// TIA Portal V17 export
// export: Created 2022-02-03T14:45:12.3278315Z, ExportSetting WithDefaults, DisplayName Totally Integrated Automation Portal, DisplayVersion V17, DisplayName TIA Portal Openness, DisplayVersion V17, DisplayName TIA Portal Version Control Interface, DisplayVersion V17, DisplayName SINAMICS Startdrive Advanced, DisplayVersion V17, DisplayName SINAMICS Startdrive G130, G150, S120, S150, SINAMICS MV, S210, DisplayVersion V17, DisplayName SINAMICS Startdrive G110M, G120, G120C, G120D, G120P, G115D, DisplayVersion V17, DisplayName STEP 7 Professional, DisplayVersion V17, DisplayName STEP 7 Safety, DisplayVersion V17, DisplayName WinCC Advanced, DisplayVersion V17
FUNCTION_BLOCK "ConveyorWeights"   // FB4, LAD
VERSION : 0.1
// stored: Access Published, AutoNumber true, IsIECCheckEnabled false, IsRetainMemResEnabled false, MemoryReserve 100, SetENOAutomatically false, UDAEnableTagReadback false
   VAR_INPUT
      weightSimulation : UInt;
      bLightBarrier : Bool;
      conveyorLeft : Bool;
      occupiedBay : Array["FIRSTBAY".."LASTBAY"] of Bool;
   END_VAR
   VAR_OUTPUT
      weightLightBarrier : UInt;
      weightBay : Array["FIRSTBAY".."LASTBAY"] of UInt;
   END_VAR
   VAR_IN_OUT
      weightConveyor : UInt;
   END_VAR
   VAR
      statOldbLightBarrier : Bool;
      statOldOccupiedBay : Array["FIRSTBAY".."LASTBAY"] of Bool;
      InstIEC_Timer1 { S7_SetPoint := 'True'} : TON_TIME;
      InstIEC_Timer2 { S7_SetPoint := 'True'} : TON_TIME;
      InstIEC_Timer3 { S7_SetPoint := 'True'} : TON_TIME;
   END_VAR
   VAR_TEMP   // added for the SCL form of the ladder/FBD networks
      _w1 : Bool;
   END_VAR
BEGIN

REGION Network 1
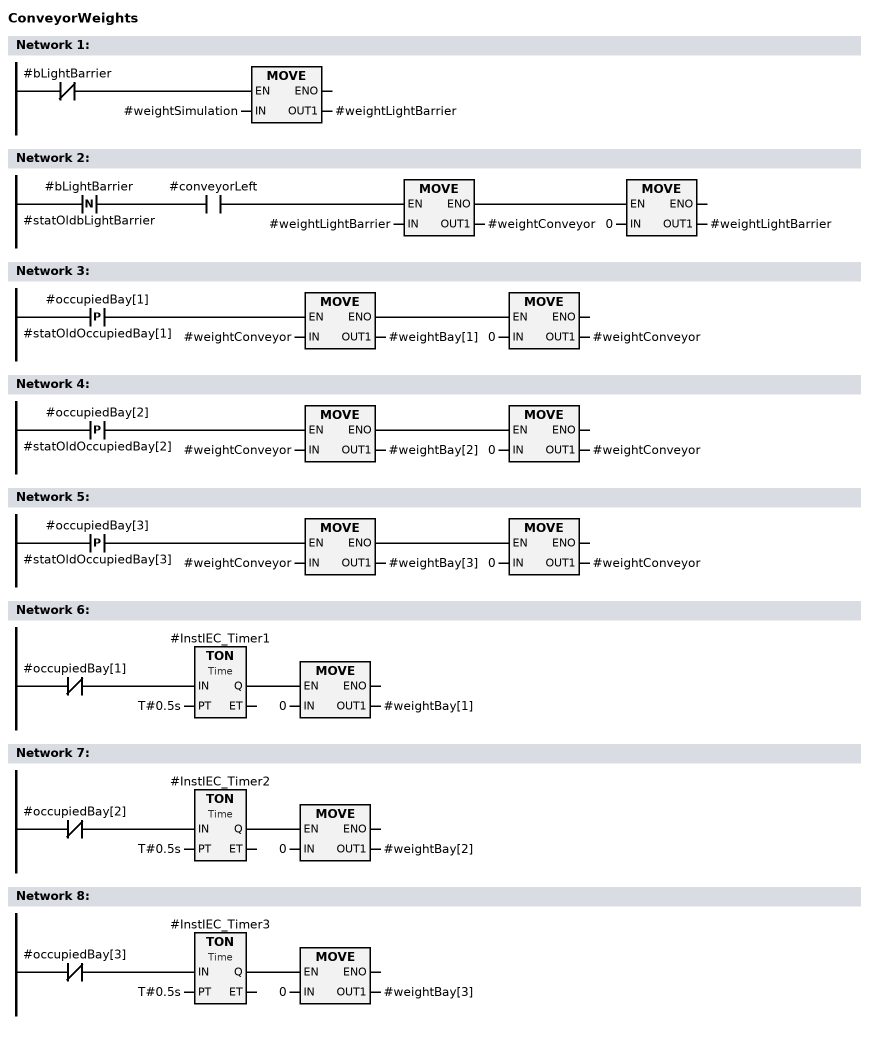
   RUNG wire#powerrail
      I_Contact( #bLightBarrier )
      Move(in := #weightSimulation, out1 => #weightLightBarrier)
   END_RUNG
   // the same network as SCL:
   IF NOT #bLightBarrier THEN #weightLightBarrier := #weightSimulation; END_IF;
END_REGION

REGION Network 2
   RUNG wire#powerrail
      N_Contact(operand := #bLightBarrier, bit := #statOldbLightBarrier)
      Contact( #conveyorLeft )
      Move(in := #weightLightBarrier, out1 => #weightConveyor)
      Move(in := 0, out1 => #weightLightBarrier)
   END_RUNG
   // the same network as SCL:
   #_w1 := NOT #bLightBarrier AND #statOldbLightBarrier;   // falling edge of #bLightBarrier
   #statOldbLightBarrier := #bLightBarrier;
   IF #_w1 AND #conveyorLeft THEN
       #weightConveyor := #weightLightBarrier;
       #weightLightBarrier := 0;
   END_IF;
END_REGION

REGION Network 3
   RUNG wire#powerrail
      P_Contact(operand := #occupiedBay[1], bit := #statOldOccupiedBay[1])
      Move(in := #weightConveyor, out1 => #weightBay[1])
      Move(in := 0, out1 => #weightConveyor)
   END_RUNG
   // the same network as SCL:
   #_w1 := #occupiedBay[1] AND NOT #statOldOccupiedBay[1];   // rising edge of #occupiedBay[1]
   #statOldOccupiedBay[1] := #occupiedBay[1];
   IF #_w1 THEN
       #weightBay[1] := #weightConveyor;
       #weightConveyor := 0;
   END_IF;
END_REGION

REGION Network 4
   RUNG wire#powerrail
      P_Contact(operand := #occupiedBay[2], bit := #statOldOccupiedBay[2])
      Move(in := #weightConveyor, out1 => #weightBay[2])
      Move(in := 0, out1 => #weightConveyor)
   END_RUNG
   // the same network as SCL:
   #_w1 := #occupiedBay[2] AND NOT #statOldOccupiedBay[2];   // rising edge of #occupiedBay[2]
   #statOldOccupiedBay[2] := #occupiedBay[2];
   IF #_w1 THEN
       #weightBay[2] := #weightConveyor;
       #weightConveyor := 0;
   END_IF;
END_REGION

REGION Network 5
   RUNG wire#powerrail
      P_Contact(operand := #occupiedBay[3], bit := #statOldOccupiedBay[3])
      Move(in := #weightConveyor, out1 => #weightBay[3])
      Move(in := 0, out1 => #weightConveyor)
   END_RUNG
   // the same network as SCL:
   #_w1 := #occupiedBay[3] AND NOT #statOldOccupiedBay[3];   // rising edge of #occupiedBay[3]
   #statOldOccupiedBay[3] := #occupiedBay[3];
   IF #_w1 THEN
       #weightBay[3] := #weightConveyor;
       #weightConveyor := 0;
   END_IF;
END_REGION

REGION Network 6
   RUNG wire#powerrail
      I_Contact( #occupiedBay[1] )
      { S7_Templates := "time_type := Time" } #InstIEC_Timer1.TON(pt := T#0.5s, et =>)
      Move(in := 0, out1 => #weightBay[1])
   END_RUNG
   // the same network as SCL:
   #InstIEC_Timer1(IN := NOT #occupiedBay[1], PT := T#0.5s);   // TON
   IF #InstIEC_Timer1.Q THEN #weightBay[1] := 0; END_IF;
END_REGION

REGION Network 7
   RUNG wire#powerrail
      I_Contact( #occupiedBay[2] )
      { S7_Templates := "time_type := Time" } #InstIEC_Timer2.TON(pt := T#0.5s, et =>)
      Move(in := 0, out1 => #weightBay[2])
   END_RUNG
   // the same network as SCL:
   #InstIEC_Timer2(IN := NOT #occupiedBay[2], PT := T#0.5s);   // TON
   IF #InstIEC_Timer2.Q THEN #weightBay[2] := 0; END_IF;
END_REGION

REGION Network 8
   RUNG wire#powerrail
      I_Contact( #occupiedBay[3] )
      { S7_Templates := "time_type := Time" } #InstIEC_Timer3.TON(pt := T#0.5s, et =>)
      Move(in := 0, out1 => #weightBay[3])
   END_RUNG
   // the same network as SCL:
   #InstIEC_Timer3(IN := NOT #occupiedBay[3], PT := T#0.5s);   // TON
   IF #InstIEC_Timer3.Q THEN #weightBay[3] := 0; END_IF;
END_REGION
END_FUNCTION_BLOCK
